FUNCTION_BLOCK FB_ManualControl_1 IMPLEMENTS  I_ManualControl
VAR_INPUT
END_VAR
VAR_OUTPUT
END_VAR
VAR
	TEMP_1 : BOOL;
	Counter : INT;
	TEMP : BOOL;

	
END_VAR

{warning 'add method implementation '}
METHOD M_RunPump : BOOL
VAR_INPUT
	bStart	: BOOL;
	NTimes : INT;

END_VAR
VAR
	
END_VAR

IF NTimes <> 0 THEN
	IF TRUE THEN
	Counter := Counter + 1;
	END_IF
	IF Counter >= (100/(2*NTimes)) THEN
		TEMP := TRUE;
	ELSE
		TEMP := FALSE;
	END_IF
	IF Counter >= (200/(2*NTimes)) THEN
		Counter := 0;
	END_IF
ELSE
	RETURN;
END_IF

IF bstart THEN
	M_RunPump := TEMP;
ELSE
	M_RunPump := FALSE;
END_IF
END_METHOD

{warning 'add method implementation '}
METHOD M_RunValve : BOOL
VAR_INPUT
	bStart	: BOOL;
END_VAR
VAR
	
END_VAR
M_RunValve := bStart;
END_METHOD

END_FUNCTION_BLOCK

(* stored: Version 1.1.0.1, ProductVersion 3.1.4024.5
   POU FB_ManualControl_1: Id {713584f3-8ee5-4aeb-86fc-744dcb4914cf}, SpecialFunc None
   Method M_RunPump: Id {143d5c78-d854-4d14-a8a0-894e56593f3f}
   Method M_RunValve: Id {2879ea4d-dcfb-4ea7-82d5-a5d34e3e8e6a} *)
